FUNCTION_BLOCK OUT_ARRAY (* ARRAY Output to TextField *)
  (* Standard: 61499-1; Classification: GUI *)
  (* Version 0.3, 2002-05-03, JHC, Rockwell Automation, Made QI IV=true. *)
  (* Version 0.2, 2001-06-01, JHC, Rockwell Automation, Added W input to subclass from OUT_ANY. *)
  (* Version 0.1, 2001-05-27, JHC, Rockwell Automation, XML version with N,TYPE inputs *)
  (* Version 0.0, 1998-12-30, JHC, Rockwell Automation, Original SRC version *)
  (* Compiler header: package fb.rt.net; *)
  (* Compiler Java IBM VisualAge 3.0 *)
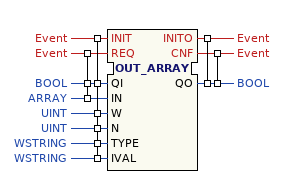
  EVENT_INPUT
    INIT WITH QI, W, N, TYPE, IVAL; (* Initialization *)
    REQ WITH QI, IN; (* Request *)
  END_EVENT
  EVENT_OUTPUT
    INITO WITH QO; (* Initialization Confirm *)
    CNF WITH QO; (* Service Confirmation *)
  END_EVENT
  VAR_INPUT
    QI : BOOL := true; (* Input event qualifier *)
    IN : ARRAY; (* Output value *)
    W : UINT := 20; (* TextField width in chars *)
    N : UINT; (* Number of array elements *)
    TYPE : WSTRING; (* Array element type *)
    IVAL : WSTRING; (* Initial contents *)
  END_VAR
  VAR_OUTPUT
    QO : BOOL; (* Output event qualifier *)
  END_VAR
END_FUNCTION_BLOCK
